# EPICS autosave request: iocs/PhotonII_IOC/iocBoot/iocPhotonII/auto_settings.req
file "PhotonII_settings.req",     P=$(P),  R=cam1:
file "NDStdArrays_settings.req",  P=$(P),  R=image1:
file "commonPlugin_settings.req", P=$(P)
